ADAPTER PICKER_SI (* Adapter Interface for Picker module *)
  (* Standard: 61499-1 *)
  (* Version 0.2, 2003-12-05, JHC, Rockwell Automation, Changed name from NEWADAPTER *)
  (* Version 0.1, 2002-01-08, JHC, Rockwell Automation, Added IND/RSP, renamed data, added sequences. *)
  (* Version 0.0, 2000-05-27, JHC, Rockwell Automation *)
  (* Compiler header: package fb.rt.pnp; *)
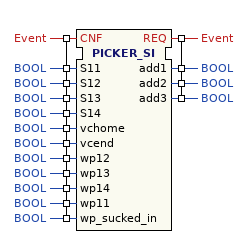
  EVENT_INPUT
    CNF WITH S11, S12, S13, S14, vchome, vcend, wp12, wp13, wp14, wp11, wp_sucked_in; (* Confirmation from Plug *)
  END_EVENT
  EVENT_OUTPUT
    REQ WITH add1, add2, add3; (* Request from Socket *)
  END_EVENT
  VAR_INPUT
    S11 : BOOL;
    S12 : BOOL;
    S13 : BOOL;
    S14 : BOOL;
    vchome : BOOL;
    vcend : BOOL;
    wp12 : BOOL;
    wp13 : BOOL;
    wp14 : BOOL;
    wp11 : BOOL;
    wp_sucked_in : BOOL;
  END_VAR
  VAR_OUTPUT
    add1 : BOOL;
    add2 : BOOL;
    add3 : BOOL;
  END_VAR
  SERVICE SOCKET/PLUG
    SEQUENCE request_confirm
      SOCKET.REQ(REQD) -> PLUG.REQ(REQD);
      PLUG.CNF(CNFD) -> SOCKET.CNF(CNFD);
    END_SEQUENCE
    SEQUENCE indication_response
      PLUG.IND(INDD) -> SOCKET.IND(INDD);
      SOCKET.RSP(RSPD) -> PLUG.RSP(RSPD);
    END_SEQUENCE
  END_SERVICE
END_ADAPTER
